# EPICS substitutions: mpgSupport/Db/ioc/edefSimSys3.substitutions
# one per system - declare EVG stuff in this IOC for testing

file bsaEdefAll.db {
  pattern { SYSI  , DEVICE        , CARDI , CHECKI }
 	  { SYS3  , IOC:SYS3:1    ,   0   ,    0   }
}
file evrPatternAll.db {
#	    Device     ,          PNET Processing
  pattern { DEVICE     , LINK4 ,      LINK5        ,      LINK6          , LINKD }
	  { IOC:SYS3:1 ,  ""   , "IOC:SYS3:1:PNET" , "IOC:SYS3:1:EDEFFO" ,  ""   }
}
file mpgPatternTest.db {
  pattern { SYSI  , UNITI }
 	  { SYS3  ,  1    }
}
